// TIA Portal V20 export
DATA_BLOCK "Ref"   // DB600
{ S7_Optimized_Access := 'TRUE' }
// stored: AutoNumber false, IsRetainMemResEnabled true, MemoryReserve 500, RetainMemoryReserve 500
   VAR RETAIN
      adjTopCalOffset : DInt := -300;   // adjustment top calibration offset [mm/10]
      adjLeftCalOffset : DInt := 150;   // adjustment left calibration offset [mm/10]
      adjRightCalOffset : DInt := 101;   // adjustment right calibration offset [mm/10]
      adjScannerTar : Real := 60.0;   // adjustment scanner target position [mm/10]
      adjTopTar : Real := 12.0;   // adjustment top target position [mm/10]
      adjLeftTar : Real := 87.5;   // adjustment left target position [mm/10]
      adjRightTar : Real := 82.6;   // adjustment right target position [mm/10]
      adjScannerAct : DInt := -2135;   // adjustment scanner target position [mm/10]
      adjTopAct : DInt := -30;   // adjustment top target position [mm/10]
      adjLeftAct : DInt := 825;   // adjustment left target position [mm/10]
      adjRightAct : DInt := 825;   // adjustment right target position [mm/10]
      senTopCalOffset : Real := 0.0;   // sensor top calibration offset [mm]
      senLeftCalOffset : Real := 0.0;   // sensor left calibration offset [mm]
      senRightCalOffset : Real := 0.0;   // sensor right calibration offset [mm]
   END_VAR
BEGIN
END_DATA_BLOCK
